// TIA Portal V19 export
DATA_BLOCK "A0303_TraslazioneStrato_PERS"   // DB103
// stored: MemoryReserve 100
   VAR RETAIN
      Par : Struct
         Ax_Man : "Positioning_EPOS_Machine_Par";
         Ax_Aut { ExternalAccessible := 'False'; ExternalVisible := 'False'; ExternalWritable := 'False'} : "Mach_Speed_Par";
         ToleranceHeight : LReal := 15.0;
         TimeoutTolerance : Time := T#0MS;
         Pers_Data_Testa : Struct
            EncoderAbsolute_Preset_OK : Bool := TRUE;
            Persistent_ActualPosition : LReal := -999.971;
         END_STRUCT;
         Pers_Data_Coda : Struct
            EncoderAbsolute_Preset_OK : Bool := TRUE;
            Persistent_ActualPosition : LReal := -999.973;
         END_STRUCT;
         Sens_Testa : "Analogic_SensorManagement_Par";
         Sens_Coda : "Analogic_SensorManagement_Par";
      END_STRUCT;
      Data_Testa : "Analogic_SensorManagement_Data";
      Data_Coda : "Analogic_SensorManagement_Data";
      Par_Mach : Struct
         PosPrelievo : LReal := -1000.0;
         PosDeposito : LReal := 5.0;
         ToleranceWindow : LReal := 0.7;
      END_STRUCT;
   END_VAR
BEGIN
   Par.Ax_Man.PosTolerance := 1.0;
   Par.Ax_Man.DelayInPosition := T#200MS;
   Par.Ax_Man.Man_Vel := 20000.0;
   Par.Ax_Man.Man_Acc := 1000.0;
   Par.Ax_Man.Man_Dec := 250.0;
   Par.Ax_Aut.SemiAut_Vel := 10000.0;
   Par.Ax_Aut.Aut_Vel := 15000.0;
   Par.Ax_Aut.Aut_Acc := 1000.0;
   Par.Ax_Aut.Aut_Dec := 1000.0;
   Par.Sens_Testa.Enable := TRUE;
   Par.Sens_Testa.RangeLow := -65.0;
   Par.Sens_Testa.RangeHigh := 35.0;
   Par.Sens_Coda.Enable := TRUE;
   Par.Sens_Coda.RangeLow := -65.0;
   Par.Sens_Coda.RangeHigh := 35.0;
   Data_Testa.OffsetValue := 20.6033496856689;
   Data_Testa.OffsetValid := TRUE;
   Data_Coda.OffsetValue := 17.6851005554199;
   Data_Coda.OffsetValid := TRUE;
END_DATA_BLOCK
